FUNCTION F_LogInfo : STRING;
VAR_INPUT
   Message : T_MaxString;
END_VAR

F_LogInfo := F_Logger(ADSLOG_MSGTYPE_HINT, Message);

END_FUNCTION

(* stored: Version 1.1.0.1, ProductVersion 3.1.4026.12
   POU F_LogInfo: Id {b101d792-3c68-0bbf-00de-22e6617441b1}, SpecialFunc None *)
